  gc_DbmTranslation_de_Text2121 : WSTRING(91) := "Turret negative end stop threshold use to reduce speed (relative to the end stop threshold)";
  gc_DbmTranslation_de_Text2122 : WSTRING(34) := "Turret positive end stop threshold";
  gc_DbmTranslation_de_Text2123 : WSTRING(56) := "Turret positive end stop threshold hysteresis (relative)";
  gc_DbmTranslation_de_Text2124 : WSTRING(91) := "Turret positive end stop threshold use to reduce speed (relative to the end stop threshold)";
  gc_DbmTranslation_de_Text2125 : WSTRING(32) := "Folded Delta arm angle threshold";
  gc_DbmTranslation_de_Text2126 : WSTRING(48) := "Folded Delta arm threshold hysteresis (relative)";
  gc_DbmTranslation_de_Text2127 : WSTRING(92) := "Delta arm bottom end stop threshold use to reduce speed (relative to the end stop threshold)";
  gc_DbmTranslation_de_Text2128 : WSTRING(32) := "Delta arm top end stop threshold";
  gc_DbmTranslation_de_Text2129 : WSTRING(54) := "Delta arm top end stop threshold hysteresis (relative)";
  gc_DbmTranslation_de_Text2130 : WSTRING(89) := "Delta arm top end stop threshold use to reduce speed (relative to the end stop threshold)";
  gc_DbmTranslation_de_Text2131 : WSTRING(32) := "Folded Delta arm angle threshold";
  gc_DbmTranslation_de_Text2132 : WSTRING(57) := "Arrow arm bottom end stop threshold hysteresis (relative)";
  gc_DbmTranslation_de_Text2133 : WSTRING(67) := "Down Delta arm slow speed reduc when delta arm is close at abutment";
  gc_DbmTranslation_de_Text2134 : WSTRING(44) := "Arrow Arm at the Top End Stop Slow Threshold";
  gc_DbmTranslation_de_Text2135 : WSTRING(40) := "Arrow Arm Bottom End Stop Slow Threshold";
  gc_DbmTranslation_de_Text2136 : WSTRING(32) := "Arrow Arm Top End Stop Threshold";
  gc_DbmTranslation_de_Text2137 : WSTRING(32) := "Arrow Arm Slow Mvt Down End Stop";
  gc_DbmTranslation_de_Text2138 : WSTRING(30) := "Arrow Arm Slow Mvt Up End Stop";
  gc_DbmTranslation_de_Text2139 : WSTRING(34) := "Telescope Slow Mvt Folded End Stop";
  gc_DbmTranslation_de_Text2140 : WSTRING(33) := "Thres of maximum Telescope sector";
  gc_DbmTranslation_de_Text2141 : WSTRING(40) := "Hyst of thres to the sector of Telescope";
  gc_DbmTranslation_de_Text2142 : WSTRING(42) := "Thres for the slow sector to the Telescope";
  gc_DbmTranslation_de_Text2143 : WSTRING(34) := "Rear center position of the turret";
  gc_DbmTranslation_de_Text2144 : WSTRING(61) := "Front center position of the turret in the positive direction";
  gc_DbmTranslation_de_Text2145 : WSTRING(61) := "Front center position of the turret in the negative direction";
  gc_DbmTranslation_de_Text2146 : WSTRING(60) := "Turret center zone window (relative to the center positions)";
  gc_DbmTranslation_de_Text2147 : WSTRING(62) := "Hysteresis applied to the turret center zone window (relative)";
  gc_DbmTranslation_de_Text2148 : WSTRING(93) := "Threshold use to reduce speed before reaching a center zone (relative to the center position)";
  gc_DbmTranslation_de_Text2149 : WSTRING(66) := "Turret center zone window left  (relative to the center positions)";
  gc_DbmTranslation_de_Text2150 : WSTRING(66) := "Turret center zone window right (relative to the center positions)";
  gc_DbmTranslation_de_Text2151 : WSTRING(33) := "Stop the basket rotation movement";
  gc_DbmTranslation_de_Text2152 : WSTRING(33) := "Stop the turret rotation movement";
  gc_DbmTranslation_de_Text2153 : WSTRING(49) := "Reduce the speed of the turret clockwise movement";
  gc_DbmTranslation_de_Text2154 : WSTRING(57) := "Reduce the speed of the turret counter clockwise movement";
  gc_DbmTranslation_de_Text2155 : WSTRING(30) := "Turret is in a center position";
  gc_DbmTranslation_de_Text2156 : WSTRING(80) := "Enable simulation mode (use the simulation variables instead of the real inputs)";
  gc_DbmTranslation_de_Text2157 : WSTRING(54) := "Test variable for simulation - basket left side sensor";
  gc_DbmTranslation_de_Text2158 : WSTRING(55) := "Test variable for simulation - basket right side sensor";
  gc_DbmTranslation_de_Text2159 : WSTRING(82) := "Test variable for simulation - a command for the rotation of the basket is enabled";
  gc_DbmTranslation_de_Text2160 : WSTRING(54) := "Test variable for simulation - turret angular position";
  gc_DbmTranslation_de_Text2161 : WSTRING(82) := "Test variable for simulation - a command for the rotation of the turret is enabled";
  gc_DbmTranslation_de_Text2162 : WSTRING(33) := "Turret is in the rear center zone";
  gc_DbmTranslation_de_Text2163 : WSTRING(43) := "Turret is in the front positive center zone";
  gc_DbmTranslation_de_Text2164 : WSTRING(43) := "Turret is in the front negative center zone";
  gc_DbmTranslation_de_Text2165 : WSTRING(26) := "Basket in centrer position";
  gc_DbmTranslation_de_Text2166 : WSTRING(31) := "Turret rotation command enabled";
  gc_DbmTranslation_de_Text2167 : WSTRING(38) := "counter stop turret rotation for debug";
  gc_DbmTranslation_de_Text2168 : WSTRING(41) := "counter no stop turret rotation for debug";
  gc_DbmTranslation_de_Text2169 : WSTRING(63) := "Fonction active when commande neutre and button fucntion pushed";
  gc_DbmTranslation_de_Text2170 : WSTRING(61) := "Command neutre when all command of TOR movement is not pushed";
  gc_DbmTranslation_de_Text2171 : WSTRING(74) := "Authorize driving mast when fonction active and dead man pedal are actived";
  gc_DbmTranslation_de_Text2172 : WSTRING(23) := "Folded position of mast";
  gc_DbmTranslation_de_Text2173 : WSTRING(45) := "Stop all movement TOR when mast is sollicited";
  gc_DbmTranslation_de_Text2174 : WSTRING(28) := "Raz distance traveled button";
  gc_DbmTranslation_de_Text2175 : WSTRING(30) := "Distance traveled in milimeter";
  gc_DbmTranslation_de_Text2176 : WSTRING(46) := "Delta beetween min and max encodeur mast value";
  gc_DbmTranslation_de_Text2177 : WSTRING(48) := "Mast measure encodeur in cm additional to offset";
  gc_DbmTranslation_de_Text2178 : WSTRING(27) := "Mast measure encodeur in cm";
  gc_DbmTranslation_de_Text2179 : WSTRING(21) := "No movement is during";
  gc_DbmTranslation_de_Text2180 : WSTRING(71) := "Scaling joystick mat , joytstick telescope is used to pilot mat measure";
  gc_DbmTranslation_de_Text2181 : WSTRING(25) := "Time with mast not folded";
  gc_DbmTranslation_de_Text2182 : WSTRING(56) := "Down axle oscillant when function mast measure is active";
  gc_DbmTranslation_de_Text2183 : WSTRING(58) := "Flag to disply on scree distance traveled wth unfolded mat";
  gc_DbmTranslation_de_Text2184 : WSTRING(22) := "Mast in upper position";
  gc_DbmTranslation_de_Text2185 : WSTRING(23) := "Mast in folded position";
  gc_DbmTranslation_de_Text2186 : WSTRING(27) := "Mast valve en down position";
  gc_DbmTranslation_de_Text2187 : WSTRING(31) := "Post interdiction for mast SNCF";
  gc_DbmTranslation_de_Text2188 : WSTRING(38) := "Memorisation of first valid cycle mast";
  gc_DbmTranslation_de_Text2189 : WSTRING(33) := "Mast contact autorisation of mvts";
  gc_DbmTranslation_de_Text2190 : WSTRING(39) := "Interdiction of Nacelle And Turret post";
  gc_DbmTranslation_de_Text2191 : WSTRING(52) := "Warning picto for the first valid cycle of mast SNCF";
  gc_DbmTranslation_de_Text2192 : WSTRING(53) := "offset mast in centimeter additional to scaling value";
  gc_DbmTranslation_de_Text2193 : WSTRING(19) := "Folded mat treshold";
  gc_DbmTranslation_de_Text2194 : WSTRING(30) := "Folded mat treshold hysterisys";
  gc_DbmTranslation_de_Text2195 : WSTRING(51) := "Min calibration value of encodeut mast sensor value";
  gc_DbmTranslation_de_Text2196 : WSTRING(51) := "Max calibration value of encodeut mast sensor value";
  gc_DbmTranslation_de_Text2197 : WSTRING(52) := "Min calibration value of encodeut mast in centimeter";
  gc_DbmTranslation_de_Text2198 : WSTRING(52) := "Max calibration value of encodeut mast in centimeter";
  gc_DbmTranslation_de_Text2199 : WSTRING(91) := "Refresh cycle time or the mast digital display ( cycle time of the message sent to display)";
  gc_DbmTranslation_de_Text2200 : WSTRING(29) := "Activate Measuring Mast (A21)";
  gc_DbmTranslation_de_Text2201 : WSTRING(76) := "Button for the calibration of min position mast measure encodeur  is pressed";
  gc_DbmTranslation_de_Text2202 : WSTRING(76) := "Button for the calibration of max position mast measure encodeur  is pressed";
  gc_DbmTranslation_de_Text2203 : WSTRING(58) := "Button for save min and max value of encodeur mast measure";
  gc_DbmTranslation_de_Text2204 : WSTRING(60) := "Raz distance translation traveled with mast measure unfolded";
  gc_DbmTranslation_de_Text2205 : WSTRING(13) := "Serial Number";
  gc_DbmTranslation_de_Text2206 : WSTRING(18) := "BP Basket Validate";
  gc_DbmTranslation_de_Text2207 : WSTRING(19) := "Key Filter Overload";
  gc_DbmTranslation_de_Text2208 : WSTRING(13) := "Key Next Mode";
  gc_DbmTranslation_de_Text2209 : WSTRING(13) := "Key Prev Mode";
  gc_DbmTranslation_de_Text2210 : WSTRING(17) := "Key Signal Danger";
  gc_DbmTranslation_de_Text2211 : WSTRING(18) := "Key Flash Light ON";
  gc_DbmTranslation_de_Text2212 : WSTRING(18) := "Key Calib Mast Min";
  gc_DbmTranslation_de_Text2213 : WSTRING(18) := "Key Calib Mast Max";
  gc_DbmTranslation_de_Text2214 : WSTRING(17) := "KeyCalibMastValid";
  gc_DbmTranslation_de_Text2215 : WSTRING(24) := "Key Generator Activation";
  gc_DbmTranslation_de_Text2216 : WSTRING(31) := "Bypass pressure threshold alarm";
  gc_DbmTranslation_de_Text2217 : WSTRING(66) := "DM_TELESCOPE_SENSOR_FAULT - Telescope In torlerance with inductive";
  gc_DbmTranslation_de_Text2218 : WSTRING(78) := "DM_TELESCOPE_SENSOR_FAULT - Telescope torlerance when no movement is solicited";
  gc_DbmTranslation_de_Text2219 : WSTRING(68) := "DM_TELESCOPE_SENSOR_FAULT - Telescope torlerance beetween 2 Channels";
  gc_DbmTranslation_de_Text2220 : WSTRING(64) := "DM__INC_ALTERNATOR_CHARGE_FAULT - max treshold alternator regime";
  gc_DbmTranslation_de_Text2221 : WSTRING(62) := "DM__INC_ALTERNATOR_CHARGE_FAULT - min treshold battery voltage";
  gc_DbmTranslation_de_Text2222 : WSTRING(108) := "DM_C1_OUT_OF_RANGE_JOY_DELTA_ARM_48XS - min alarm value of joytick delta arm in % according batterie voltage";
  gc_DbmTranslation_de_Text2223 : WSTRING(108) := "DM_C1_OUT_OF_RANGE_JOY_DELTA_ARM_48XS - max alarm value of joytick delta arm in % according batterie voltage";
  gc_DbmTranslation_de_Text2224 : WSTRING(108) := "DM_C1_OUT_OF_RANGE_JOY_ARROW_ARM_48XS - min alarm value of joytick arrow arm in % according batterie voltage";
  gc_DbmTranslation_de_Text2225 : WSTRING(108) := "DM_C1_OUT_OF_RANGE_JOY_ARROW_ARM_48XS - max alarm value of joytick arrow arm in % according batterie voltage";
  gc_DbmTranslation_de_Text2226 : WSTRING(116) := "DM_C1_OUT_OF_RANGE_JOY_TELESCOPE_ARM_48XS - min alarm value of joytick telescope arm in % according batterie voltage";
  gc_DbmTranslation_de_Text2227 : WSTRING(116) := "DM_C1_OUT_OF_RANGE_JOY_TELESCOPE_ARM_48XS - max alarm value of joytick telescope arm in % according batterie voltage";
  gc_DbmTranslation_de_Text2228 : WSTRING(123) := "DM_C1_OUT_OF_RANGE_JOY_ROT_TURRET_ARM_48XS - min alarm value of joytick rotation turret arm in % according batterie voltage";
  gc_DbmTranslation_de_Text2229 : WSTRING(123) := "DM_C1_OUT_OF_RANGE_JOY_ROT_TURRET_ARM_48XS - max alarm value of joytick rotation turret arm in % according batterie voltage";
  gc_DbmTranslation_de_Text2230 : WSTRING(120) := "DM_C1_OUT_OF_RANGE_JOY_ADVANCEMENT_48XS - min alarm value of joytick rotation turret arm in % according batterie voltage";
  gc_DbmTranslation_de_Text2231 : WSTRING(120) := "DM_C1_OUT_OF_RANGE_JOY_ADVANCEMENT_48XS - max alarm value of joytick rotation turret arm in % according batterie voltage";
  gc_DbmTranslation_de_Text2232 : WSTRING(17) := "Time Bypass Fault";
  gc_DbmTranslation_de_Text2233 : WSTRING(26) := "Timer for the Bypass fault";
  gc_DbmTranslation_de_Text2234 : WSTRING(42) := "Inconsistency Nc No logical frame rotation";
  gc_DbmTranslation_de_Text2235 : WSTRING(65) := "internal error , inconsistency between two channels and can error";
  gc_DbmTranslation_de_Text2236 : WSTRING(37) := "Fault of Ev park brake axle osccilant";
  gc_DbmTranslation_de_Text2237 : WSTRING(32) := "Fault of Ev park brake axle fixe";
  gc_DbmTranslation_de_Text2238 : WSTRING(40) := "Fault of Ev service brake axle osccilant";
  gc_DbmTranslation_de_Text2239 : WSTRING(35) := "Fault of Ev service brake axle fixe";
  gc_DbmTranslation_de_Text2240 : WSTRING(30) := "Fault of Ev serice brake track";
  gc_DbmTranslation_de_Text2241 : WSTRING(27) := "RM com can radio loss by C0";
  gc_DbmTranslation_de_Text2242 : WSTRING(33) := "Ev 2nd Park Brake Axle Fixe Fault";
  gc_DbmTranslation_de_Text2243 : WSTRING(33) := "Ev 2nd Park Brake Axle Osci Fault";
  gc_DbmTranslation_de_Text2244 : WSTRING(0) := "";
  gc_DbmTranslation_de_Text2245 : WSTRING(0) := "";
  gc_DbmTranslation_de_Text2246 : WSTRING(0) := "";
  gc_DbmTranslation_de_Text2247 : WSTRING(0) := "";
  gc_DbmTranslation_de_Text2248 : WSTRING(0) := "";
  gc_DbmTranslation_de_Text2249 : WSTRING(0) := "";
  gc_DbmTranslation_de_Text2250 : WSTRING(0) := "";
  gc_DbmTranslation_de_Text2251 : WSTRING(0) := "";
  gc_DbmTranslation_de_Text2252 : WSTRING(0) := "";
  gc_DbmTranslation_de_Text2253 : WSTRING(0) := "";
  gc_DbmTranslation_de_Text2254 : WSTRING(0) := "";
  gc_DbmTranslation_de_Text2255 : WSTRING(0) := "";
  gc_DbmTranslation_de_Text2256 : WSTRING(0) := "";
  gc_DbmTranslation_de_Text2257 : WSTRING(28) := "Additionnal Performance Func";
  gc_DbmTranslation_de_Text2258 : WSTRING(21) := "Slope Case Less 2 Deg";
  gc_DbmTranslation_de_Text2259 : WSTRING(21) := "Slope Case Less 4 Deg";
  gc_DbmTranslation_de_Text2260 : WSTRING(21) := "Slope Case Less 6 Deg";
  gc_DbmTranslation_de_Text2261 : WSTRING(23) := "Slope Case Higher 6 Deg";
  gc_DbmTranslation_de_Text2262 : WSTRING(26) := "Turret In Speed Zone 2 Deg";
  gc_DbmTranslation_de_Text2263 : WSTRING(26) := "Turret In Speed Zone 4 Deg";
  gc_DbmTranslation_de_Text2264 : WSTRING(37) := "Turret In Speed Zone 2 Deg For Basket";
  gc_DbmTranslation_de_Text2265 : WSTRING(21) := "Selected control post";
  gc_DbmTranslation_de_Text2266 : WSTRING(23) := "Mast sensor position UP";
  gc_DbmTranslation_de_Text2267 : WSTRING(40) := "Hydraulic valve uin down position sensor";
  gc_DbmTranslation_de_Text2268 : WSTRING(28) := "Measuring mast sensor folded";
  gc_DbmTranslation_de_Text2269 : WSTRING(35) := "Presence of sensor plate on machine";
  gc_DbmTranslation_de_Text2270 : WSTRING(51) := "Recovery reduction ratio for the battery protection";
  gc_DbmTranslation_de_Text2271 : WSTRING(21) := "Variable debug Neotec";
  gc_DbmTranslation_de_Text2272 : WSTRING(21) := "Variable debug Neotec";
  gc_DbmTranslation_de_Text2273 : WSTRING(21) := "Variable debug Neotec";
  gc_DbmTranslation_de_Text2274 : WSTRING(21) := "Variable debug Neotec";
  gc_DbmTranslation_de_Text2275 : WSTRING(21) := "Variable debug Neotec";
  gc_DbmTranslation_de_Text2276 : WSTRING(21) := "Variable debug Neotec";
  gc_DbmTranslation_de_Text2277 : WSTRING(21) := "Variable debug Neotec";
  gc_DbmTranslation_de_Text2278 : WSTRING(21) := "Variable debug Neotec";
  gc_DbmTranslation_de_Text2279 : WSTRING(21) := "Variable debug Neotec";
  gc_DbmTranslation_de_Text2280 : WSTRING(21) := "Variable debug Neotec";
  gc_DbmTranslation_de_Text2281 : WSTRING(21) := "Variable debug Neotec";
  gc_DbmTranslation_de_Text2282 : WSTRING(21) := "Variable debug Neotec";
  gc_DbmTranslation_de_Text2283 : WSTRING(21) := "Variable debug Neotec";
  gc_DbmTranslation_de_Text2284 : WSTRING(21) := "Variable debug Neotec";
  gc_DbmTranslation_de_Text2285 : WSTRING(21) := "Variable debug Neotec";
  gc_DbmTranslation_de_Text2286 : WSTRING(21) := "Variable debug Neotec";
  gc_DbmTranslation_de_Text2287 : WSTRING(21) := "Variable debug Neotec";
  gc_DbmTranslation_de_Text2288 : WSTRING(21) := "Variable debug Neotec";
  gc_DbmTranslation_de_Text2289 : WSTRING(21) := "Variable debug Neotec";
  gc_DbmTranslation_de_Text2290 : WSTRING(21) := "Variable debug Neotec";
  gc_DbmTranslation_de_Text2291 : WSTRING(21) := "Variable debug Neotec";
  gc_DbmTranslation_de_Text2292 : WSTRING(21) := "Variable debug Neotec";
  gc_DbmTranslation_de_Text2293 : WSTRING(21) := "Variable debug Neotec";
  gc_DbmTranslation_de_Text2294 : WSTRING(21) := "Variable debug Neotec";
  gc_DbmTranslation_de_Text2295 : WSTRING(21) := "Variable debug Neotec";
  gc_DbmTranslation_de_Text2296 : WSTRING(21) := "Variable debug Neotec";
  gc_DbmTranslation_de_Text2297 : WSTRING(21) := "Variable debug Neotec";
  gc_DbmTranslation_de_Text2298 : WSTRING(21) := "Variable debug Neotec";
  gc_DbmTranslation_de_Text2299 : WSTRING(21) := "Variable debug Neotec";
  gc_DbmTranslation_de_Text2300 : WSTRING(21) := "Variable debug Neotec";
  gc_DbmTranslation_de_Text2301 : WSTRING(21) := "Variable debug Neotec";
  gc_DbmTranslation_de_Text2302 : WSTRING(21) := "Variable debug Neotec";
  gc_DbmTranslation_de_Text2303 : WSTRING(21) := "Variable debug Neotec";
  gc_DbmTranslation_de_Text2304 : WSTRING(21) := "Variable debug Neotec";
  gc_DbmTranslation_de_Text2305 : WSTRING(21) := "Variable debug Neotec";
  gc_DbmTranslation_de_Text2306 : WSTRING(21) := "Variable debug Neotec";
  gc_DbmTranslation_de_Text2307 : WSTRING(21) := "Variable debug Neotec";
  gc_DbmTranslation_de_Text2308 : WSTRING(21) := "Variable debug Neotec";
  gc_DbmTranslation_de_Text2309 : WSTRING(21) := "Variable debug Neotec";
  gc_DbmTranslation_de_Text2310 : WSTRING(21) := "Variable debug Neotec";
  gc_DbmTranslation_de_Text2311 : WSTRING(64) := "Mesure de la température du liquide de refroidissement du moteur";
  gc_DbmTranslation_de_Text2312 : WSTRING(58) := "Pression mesuré dans le système de lubrification du moteur";
  gc_DbmTranslation_de_Text2313 : WSTRING(34) := "Vitesse actuelle du moteur calculé";
  gc_DbmTranslation_de_Text2314 : WSTRING(56) := "Courant de l'alternateur principale du moteur thermique ";
  gc_DbmTranslation_de_Text2315 : WSTRING(56) := "Etat du moteur : Motor stop, pre-start, Wram-Up,Starting";
  gc_DbmTranslation_de_Text2316 : WSTRING(40) := "Tension mesuré aux bornes de la batterie";
  gc_DbmTranslation_de_Text2317 : WSTRING(33) := "Commande de la vietesse du moteur";
  gc_DbmTranslation_de_Text2318 : WSTRING(30) := "Override Control Mode (SPN695)";
  gc_DbmTranslation_de_Text2319 : WSTRING(18) := "High pressure Oil ";
  gc_DbmTranslation_de_Text2320 : WSTRING(14) := "Warmin gActive";
  gc_DbmTranslation_de_Text2321 : WSTRING(10) := "Stop Motor";
  gc_DbmTranslation_de_Text2322 : WSTRING(27) := "Regeneration SOC at maximum";
  gc_DbmTranslation_de_Text2323 : WSTRING(61) := "Threshold maximum to autorize regeneration (Threshold of SOC)";
  gc_DbmTranslation_de_Text2324 : WSTRING(42) := "Hysteresis for regeneration of SOC maximum";
  gc_DbmTranslation_de_Text2325 : WSTRING(57) := "Number of time to refuse reloading from generator (Alarm)";
  gc_DbmTranslation_de_Text2326 : WSTRING(61) := "Number of time to refuse reloading from generator (forbidden)";
  gc_DbmTranslation_de_Text2327 : WSTRING(23) := "RPM motor maximum value";
  gc_DbmTranslation_de_Text2328 : WSTRING(23) := "RPM motor minimum value";
  gc_DbmTranslation_de_Text2329 : WSTRING(27) := "RPM for a movement with PVG";
  gc_DbmTranslation_de_Text2330 : WSTRING(27) := "RPM for a movement with TOR";
  gc_DbmTranslation_de_Text2331 : WSTRING(30) := "Hydraulic oil cold temperature";
  gc_DbmTranslation_de_Text2332 : WSTRING(42) := "Capacity of the battery in ampere per hour";
  gc_DbmTranslation_de_Text2333 : WSTRING(53) := "Number of element for the remaining regeneration time";
  gc_DbmTranslation_de_Text2334 : WSTRING(61) := "Number of times the alarm regeneration threshold was exceeded";
  gc_DbmTranslation_de_Text2335 : WSTRING(89) := "Number of times we exceeded the threshold of regeneration forbidden of the electric motor";
  gc_DbmTranslation_de_Text2336 : WSTRING(25) := "Cold Oil Tank Temperature";
  gc_DbmTranslation_de_Text2337 : WSTRING(30) := "Rpm Movements on Electric Mode";
  gc_DbmTranslation_de_Text2338 : WSTRING(37) := "Rpm Translation on Rail Electric Mode";
  gc_DbmTranslation_de_Text2339 : WSTRING(24) := "Rpm Oil Tank Temperature";
  gc_DbmTranslation_de_Text2340 : WSTRING(18) := "Rpm Electric motor";
  gc_DbmTranslation_de_Text2341 : WSTRING(12) := "Generator ON";
  gc_DbmTranslation_de_Text2342 : WSTRING(23) := "Automatic mode activate";
  gc_DbmTranslation_de_Text2343 : WSTRING(21) := "Silence mode activate";
  gc_DbmTranslation_de_Text2344 : WSTRING(21) := "Forcing mode activate";
  gc_DbmTranslation_de_Text2345 : WSTRING(24) := "Forcing regeneration Low";
  gc_DbmTranslation_de_Text2346 : WSTRING(25) := "Forcing regeneration High";
  gc_DbmTranslation_de_Text2347 : WSTRING(35) := "Remaining Regeneration time average";
  gc_DbmTranslation_de_Text2348 : WSTRING(25) := "Ask Reload With Generator";
  gc_DbmTranslation_de_Text2349 : WSTRING(27) := "Reloading With Generator On";
  gc_DbmTranslation_de_Text2350 : WSTRING(24) := "Stop regeneration by SOC";
  gc_DbmTranslation_de_Text2351 : WSTRING(24) := "Total regeneration Hours";
  gc_DbmTranslation_de_Text2352 : WSTRING(31) := "Picto Cold Oil Tank Temperature";
  gc_DbmTranslation_de_Text2353 : WSTRING(20) := "Total electric hours";
  gc_DbmTranslation_de_Text2354 : WSTRING(37) := "Picto recovery reduction ratio active";
  gc_DbVarGrpNameTranslation_de_Text2355 : WSTRING(17) := "NV_PARAMERTERS_C0";
  gc_DbVarGrpNameTranslation_de_Text2356 : WSTRING(23) := "NV_PARAM_SPEED_MAX_RAIL";
  gc_DbVarGrpNameTranslation_de_Text2357 : WSTRING(19) := "NV_PARAM_BRAKE_TEST";
  gc_DbVarGrpNameTranslation_de_Text2358 : WSTRING(28) := "NV_PARAM_RAIL_WORK_SAFETY_C0";
  gc_DbVarGrpNameTranslation_de_Text2359 : WSTRING(25) := "NV_PARAM_TRANSPORT_POS_C0";
  gc_DbVarGrpNameTranslation_de_Text2360 : WSTRING(28) := "NV_PARAM_SELECT_CONTROL_POST";
  gc_DbVarGrpNameTranslation_de_Text2361 : WSTRING(17) := "NV_PARAM_ALARM_C0";
  gc_DbVarGrpNameTranslation_de_Text2362 : WSTRING(21) := "NV_PARAM_MAST_DISPLAY";
  gc_DbVarGrpNameTranslation_de_Text2363 : WSTRING(17) := "NV_PARAMERTERS_C1";
  gc_DbVarGrpNameTranslation_de_Text2364 : WSTRING(17) := "NV_PARAM_MOTOR_C1";
  gc_DbVarGrpNameTranslation_de_Text2365 : WSTRING(31) := "NV_PARAM_LIMIT_WORK_ENVELOPE_C1";
  gc_DbVarGrpNameTranslation_de_Text2366 : WSTRING(24) := "NV_PARAM_MVT_END_STOP_C1";
  gc_DbVarGrpNameTranslation_de_Text2367 : WSTRING(21) := "NV_PARAM_AUTO_STOP_C1";
  gc_DbVarGrpNameTranslation_de_Text2368 : WSTRING(16) := "NV_PARAM_MAST_C1";
  gc_DbVarGrpNameTranslation_de_Text2369 : WSTRING(17) := "NV_PARAM_ALARM_C1";
  gc_DbVarGrpNameTranslation_de_Text2370 : WSTRING(12) := "NV_OPTION_C0";
  gc_DbVarGrpNameTranslation_de_Text2371 : WSTRING(12) := "NV_OPTION_C1";
